//{{V2}}
DATA_BLOCK DB1

AUTHOR:mh
FAMILY:nb
NAME:nb
VERSION:1.0


FB1

BEGIN

       STATUS:=W#16#0000
       FEHLER:=W#16#0000
       ST_Anlauf:=W#16#0000
       ST_Referenz:=W#16#0000
       ST_Bereit:=W#16#0000
       ST_Fehler:=W#16#0000
       ST_Busy:=W#16#0000
       ST_Test:=W#16#0000
       ST_Frei:=W#16#0000
       ST_Pause:=W#16#0000
       BEREIT:=W#16#0000
       ST_BereitAufnahme:=W#16#0000
       ST_BereitAbgabe:=W#16#0000
       ST_BereitNA:=W#16#0000
END_DATA_BLOCK
